FUNCTION_BLOCK BagOpeningStatus
VAR_INPUT
END_VAR
VAR_OUTPUT
END_VAR
VAR
	bag_status	: BagStatus;
	sensor_status	: STRING;
END_VAR

PROPERTY _bagStatus : BagStatus
GET
_bagStatus	:= bag_status;
END_GET
SET
bag_status	:= _bagStatus;
END_SET
END_PROPERTY

PROPERTY _sensor_status : STRING
GET
_sensor_status	:= sensor_status;
END_GET
SET
sensor_status	:=_sensor_status;
END_SET
END_PROPERTY

END_FUNCTION_BLOCK

(* stored: Version 1.1.0.1, ProductVersion 3.1.4024.12
   POU BagOpeningStatus: Id {72a48fb8-6f11-4a1d-8d25-a42e6fe94f8f}, SpecialFunc None
   Property _bagStatus: Id {cc5662e5-94ab-4fce-b65c-e245d9be907b}
   Get Get: Id {43025794-314b-448d-a8a0-7f53a3a332d3}
   Set Set: Id {c51c65fa-aa26-402e-8b22-9daa006dee15}
   Property _sensor_status: Id {ea2ce233-2f2f-43e1-85da-0d2cb272fd7d}
   Get Get: Id {795f57d0-0089-47b7-a0b7-4928e3fc5b6d}
   Set Set: Id {2f3aa1ff-65ce-4d47-80d4-25add53989ca} *)
